// 本代码由 S7_SCL_SRC_GEN 自动生成。author: goosy.jo@gmail.com
// 配置文件: D:/codes/AS/S7-AS/MT_Poll/MT.yaml
// 摘要: 20b655b7eee2f4d7e9bc1849f898b33a

FUNCTION_BLOCK "write_DO"
TITLE='MT写命令'
VERSION:'1.0'
AUTHOR:Goosy
NAME:writeB
FAMILY:GooLib
VAR_INPUT
  r_work_F : BOOL ;                  // 设备正常指示
  r_invalid : BOOL ;                 // 设备无效指示
  r_on_receive : BOOL ;              // 设备接收指示
  r_unit_ID : BYTE ;                 // 设备号
  r_func_code : BYTE ;               // modbus功能号
  r_length : BYTE ;                  // 接收长度
  r_B0 : BYTE ;                      // 接收字节
  r_B1 : BYTE ;                      // 接收字节
  w_work_F : BOOL ;                  // 设备正常指示
  w_invalid : BOOL ;                 // 设备无效指示
  w_on_receive : BOOL ;              // 设备接收指示
  w_unit_ID : BYTE ;                 // 设备号
  w_func_code : BYTE ;               // modbus功能号
  start_H : BYTE ;                   // 写起始高字节
  start_L : BYTE ;                   // 写起始低字节
  len_H : BYTE ;                     // 写数量高字节
  len_L : BYTE ;                     // 写数量低字节
  CH : ARRAY[1..8] OF BOOL;          // QB0 数据
  B0 AT CH : BYTE;                   // QB0 数据
END_VAR
VAR_OUTPUT
  MBAP_seq         : WORD ;          // 事务号 PLC自动填写
  MBAP_protocol    : WORD := W#16#0; // 必须为0
  MBAP_length      : WORD := W#16#8; // 长度，对读命令，通常为6
  unit_ID : BYTE := B#16#3;          // 子站地址
  func_code : BYTE := B#16#F;        // modbus 功能号，15写多个线圈
  start : INT := 0;                  // 起始地址
  length : INT := 8;                 // 数据长度
  betys : BYTE := B#16#1;            // 字节数
  data : BYTE := B#16#0;             // 数据
END_VAR
VAR_IN_OUT
  writing : BOOL;                    //正在写
END_VAR
BEGIN
IF B0 <> r_B0 THEN
  data := B0;
  writing := TRUE;
END_IF;
END_FUNCTION_BLOCK

DATA_BLOCK "EDO01" "write_DO"
BEGIN
END_DATA_BLOCK


// 设备数据接收DB块，可根据设备定义多个接收DB块
// 本例DB52，在其中定义了4个设备的数据，应依据实际增减
// 建议一个设备只定义在一个DB中，本例一个DB定义多个设备仅为了展示可以这样组织
DATA_BLOCK "rdata"
STRUCT
    workOK0 : BOOL ;                 //通讯正确指示符  ===第1个接收数据 0
    invalid0 : BOOL ;                //数据无效标志
    on_receive0 : BOOL ;             //新收数据标志
    unit_ID0 : BYTE ;                //设备号
    func_code0 : BYTE ;              //modbus功能号
    length0 : BYTE ;                 //数据长度
    data0 : ARRAY[0..59] OF BYTE ;   //数据
    workOK1 : BOOL ;                 //通讯正确指示符  ===第2个接收数据 64
    invalid1 : BOOL ;                //数据无效标志
    on_receive1 : BOOL ;             //新收数据标志
    unit_ID1 : BYTE ;                //设备号
    func_code1 : BYTE ;              //modbus功能号
    length1 : BYTE ;                 //数据长度
    data1 : ARRAY[0..59] OF BYTE ;   //数据
END_STRUCT ;
BEGIN
END_DATA_BLOCK

// 连接数据块，为"MT_Poll"的背景数据块
// 一个连接就要定义一个这样的背景块。本例展示2个连接："MT01" "MT02"，依据实际增减
DATA_BLOCK "MT01" "MT_Poll" // 连接1 192.168.28.62:502
BEGIN
    TCON_Parameters.block_length := W#16#40;     //固定为64
    TCON_Parameters.id := W#16#0001;             //连接ID 每个连接必须不一样！
    TCON_Parameters.connection_type := B#16#11;  //连接类型 11H=TCP/IP native, 12H=ISO on TCP, 13H=UDP, 01=TCP/IP comp
    TCON_Parameters.active_est := TRUE;          //是否主动（本功能调用必须为TRUE）
    TCON_Parameters.local_device_id := B#16#02;  //CPU31x-2_PN/DP
    TCON_Parameters.local_tsap_id_len := B#16#0;
    TCON_Parameters.rem_subnet_id_len := B#16#0;
    TCON_Parameters.rem_staddr_len := B#16#4;
    TCON_Parameters.rem_tsap_id_len := B#16#2;
    TCON_Parameters.next_staddr_len := B#16#0;
    TCON_Parameters.rem_staddr[1] := B#16#C0;    //IP1 192
    TCON_Parameters.rem_staddr[2] := B#16#A8;    //IP2 168
    TCON_Parameters.rem_staddr[3] := B#16#1C;    //IP3 28
    TCON_Parameters.rem_staddr[4] := B#16#3E;    //IP4 62
    TCON_Parameters.rem_tsap_id[1] := B#16#01;   //PortH 502
    TCON_Parameters.rem_tsap_id[2] := B#16#F6;   //PortL
    TCON_Parameters.spare := W#16#0;             //固定为0
END_DATA_BLOCK

DATA_BLOCK "MT02" "MT_Poll" // 连接1 192.168.15.43:503
BEGIN
    TCON_Parameters.block_length := W#16#40;     //固定为64
    TCON_Parameters.id := W#16#0002;             //连接ID 每个连接必须不一样！
    TCON_Parameters.connection_type := B#16#11;  //连接类型 11H=TCP/IP native, 12H=ISO on TCP, 13H=UDP, 01=TCP/IP comp
    TCON_Parameters.active_est := TRUE;          //是否主动（本功能调用必须为TRUE）
    TCON_Parameters.local_device_id := B#16#02;  //CPU31x-2_PN/DP
    TCON_Parameters.local_tsap_id_len := B#16#0;
    TCON_Parameters.rem_subnet_id_len := B#16#0;
    TCON_Parameters.rem_staddr_len := B#16#4;
    TCON_Parameters.rem_tsap_id_len := B#16#2;
    TCON_Parameters.next_staddr_len := B#16#0;
    TCON_Parameters.rem_staddr[1] := B#16#C0;    //IP1 192
    TCON_Parameters.rem_staddr[2] := B#16#A8;    //IP2 168
    TCON_Parameters.rem_staddr[3] := B#16#0F;    //IP3 15
    TCON_Parameters.rem_staddr[4] := B#16#2B;    //IP4 43
    TCON_Parameters.rem_tsap_id[1] := B#16#01;   //PortH 503
    TCON_Parameters.rem_tsap_id[2] := B#16#F7;   //PortL
    TCON_Parameters.spare := W#16#0;             //固定为0
END_DATA_BLOCK

// 轮询定义数据块 "MT_polls_DB" DB51
// 每个TCP连接对应一个轮询序列，可以定义多个轮询序列。
// 本例只定义了2个轮询序列，即 "Poll_DB".pollList1 "Poll_DB".pollList2
// 在本块只，只能定义 01 02 03 04 05 06 功能码的数据
// 15 16 功能码的数据必须定义在其它块上
DATA_BLOCK "MT_polls_DB"
TITLE = "轮询定义"
VERSION : 0.0
STRUCT
    pollList1 : ARRAY  [0 .. 1] OF // ===== 轮询列表 连接1 192.168.28.62:502
    STRUCT
        enable         : BOOL := TRUE;  // 允许本poll通讯
        timeout        : BOOL ;         // 本 poll 通讯超时
        cyclicity      : BOOL := TRUE;  // 自动周期性触发询问，默认为TRUE，为 FALSE 时由下方手动触发
        custom_trigger : BOOL ;         // 手动触发询问
        try_times      : INT := 10;     // 最多询问失败次数，超过该次数标记该设备数据无效
        send_DB        : INT ;          // 发送DB，为0时为本块
        send_start     : INT ;          // 发送DB起始地址
        recv_DB        : INT ;          // 接收数据块号
        recv_start     : INT ;          // 接收数据块起始地址
        status         : WORD ;         // 状态
        wait_count     : INT ;          // 等待计时
    END_STRUCT ;
    pollList2 : ARRAY  [0 .. 1] OF // ===== 轮询列表 连接1 192.168.15.43:503
    STRUCT
        enable         : BOOL := TRUE;  // 允许本poll通讯
        timeout        : BOOL ;         // 本 poll 通讯超时
        cyclicity      : BOOL := TRUE;  // 自动周期性触发询问，默认为TRUE，为 FALSE 时由下方手动触发
        custom_trigger : BOOL ;         // 手动触发询问
        try_times      : INT := 10;     // 最多询问失败次数，超过该次数标记该设备数据无效
        send_DB        : INT ;          // 发送DB，为0时为本块
        send_start     : INT ;          // 发送DB起始地址
        recv_DB        : INT ;          // 接收数据块号
        recv_start     : INT ;          // 接收数据块起始地址
        status         : WORD ;         // 状态
        wait_count     : INT ;          // 等待计时
    END_STRUCT ;
    p0_data : STRUCT
        MBAP_seq : WORD ;               // 事务号 PLC自动填写
        MBAP_protocol : WORD ;          // 必须为0
        MBAP_length : WORD  := W#16#6;  // 长度，对读命令，通常为6
        unit_ID : BYTE ;                // 设备号，不关心的情况下可以填0
        func_code : BYTE ;              // modbus功能号
        address : WORD ;                // 起始地址
        data : WORD ;                   // 数据，对 05 06 功能码来说为写入值，对其它功能码来说为长度
    END_STRUCT;
    p1_data : STRUCT
        MBAP_seq : WORD ;               // 事务号 PLC自动填写
        MBAP_protocol : WORD ;          // 必须为0
        MBAP_length : WORD  := W#16#6;  // 长度，对读命令，通常为6
        unit_ID : BYTE ;                // 设备号，不关心的情况下可以填0
        func_code : BYTE ;              // modbus功能号
        address : WORD ;                // 起始地址
        data : WORD ;                   // 数据，对 05 06 功能码来说为写入值，对其它功能码来说为长度
    END_STRUCT;
    p2_data : STRUCT
        MBAP_seq : WORD ;               // 事务号 PLC自动填写
        MBAP_protocol : WORD ;          // 必须为0
        MBAP_length : WORD  := W#16#6;  // 长度，对读命令，通常为6
        unit_ID : BYTE ;                // 设备号，不关心的情况下可以填0
        func_code : BYTE ;              // modbus功能号
        address : WORD ;                // 起始地址
        data : WORD ;                   // 数据，对 05 06 功能码来说为写入值，对其它功能码来说为长度
    END_STRUCT;
END_STRUCT ;
BEGIN
    // --- 连接1 192.168.28.62:502
    // 出站1#流量计
    pollList1[0].cyclicity  := TRUE;
    pollList1[0].try_times := 10;
    pollList1[0].send_DB := 20;
    pollList1[0].send_start := 64;
    pollList1[0].recv_DB := 52;
    pollList1[0].recv_start := 0;
    // send data
    p0_data.MBAP_protocol := W#16#00;
    p0_data.MBAP_length := W#16#6;
    p0_data.unit_ID := B#16#01;
    p0_data.func_code := B#16#03;
    p0_data.address := W#16#0000;
    p0_data.data := W#16#001C;
    // 通讯状态信息
    pollList1[1].cyclicity  := TRUE;
    pollList1[1].try_times := 10;
    pollList1[1].send_DB := 20;
    pollList1[1].send_start := 76;
    pollList1[1].recv_DB := 52;
    pollList1[1].recv_start := 64;
    // send data
    p1_data.MBAP_protocol := W#16#00;
    p1_data.MBAP_length := W#16#6;
    p1_data.unit_ID := B#16#01;
    p1_data.func_code := B#16#04;
    p1_data.address := W#16#158C;
    p1_data.data := W#16#0005;

    // --- 连接1 192.168.15.43:503
    // DO读
    pollList2[0].cyclicity  := TRUE;
    pollList2[0].try_times := 10;
    pollList2[0].send_DB := 20;
    pollList2[0].send_start := 88;
    pollList2[0].recv_DB := 31;
    pollList2[0].recv_start := 0;
    // send data
    p2_data.MBAP_protocol := W#16#00;
    p2_data.MBAP_length := W#16#6;
    p2_data.unit_ID := B#16#03;
    p2_data.func_code := B#16#01;
    p2_data.address := W#16#0000;
    p2_data.data := W#16#0008;
    // DO写
    pollList2[1].cyclicity  := FALSE;
    pollList2[1].custom_trigger := FALSE;
    pollList2[1].try_times := 10;
    pollList2[1].send_DB := 31;
    pollList2[1].send_start := 16;
    pollList2[1].recv_DB := 31;
    pollList2[1].recv_start := 6;
    // pollList2 的发送数据在其它块上，不在这里定义
END_DATA_BLOCK

// 调用
FUNCTION "MT_Loop" : VOID
// 连接1 192.168.28.62:502
"MT_Poll"."MT01" (
    data := "MT_polls_DB".pollList1);
// 扩展状态位
IF "rdata".invalid1 THEN
  "rdata".data1[0] := B#16#00;
  "rdata".data1[1] := B#16#00;
  "rdata".data1[8] := B#16#00;
  "rdata".data1[9] := B#16#00;
END_IF;

// 连接1 192.168.15.43:503
// 展示部分高级用法
"MT_Poll"."MT02" (
    interval_time := 500,
    data := "MT_polls_DB".pollList2);
"write_DO"."EDO01"(writing := MT_polls_DB.pollList2[1].custom_trigger);

// 接收块

END_FUNCTION
